FUNCTION ConcatStrings : STRING_5K
VAR_IN_OUT
	stringsArr : ARRAY[*] OF STRING_5K;
END_VAR
VAR_INPUT
	opening : STRING_5K;
	closing : STRING_5K;
	separator : STRING_5K;
END_VAR
VAR
	fullString : STRING_5K;
	i : DINT := 0;	
END_VAR

fullString := opening; //opening segment

FOR i:=LOWER_BOUND(stringsArr, 1) TO UPPER_BOUND(stringsArr, 1)-1 BY 1 DO //first element to 2nd last element
	CONCAT2(ADR(fullString), ADR(stringsArr[i]), ADR(fullString), SIZEOF(fullString));
	CONCAT2(ADR(fullString), ADR(separator), ADR(fullString), SIZEOF(fullString));
END_FOR
CONCAT2(ADR(fullString), ADR(stringsArr[UPPER_BOUND(stringsArr, 1)]), ADR(fullString), SIZEOF(fullString)); //final element

CONCAT2(ADR(fullString), ADR(closing), ADR(fullString), SIZEOF(fullString)); //closing segment

concatStrings := fullString;

END_FUNCTION

(* stored: Version 1.1.0.1, ProductVersion 3.1.4024.11
   POU ConcatStrings: Id {a680f869-5d97-4700-8d94-791d083cc0a3}, SpecialFunc None *)
